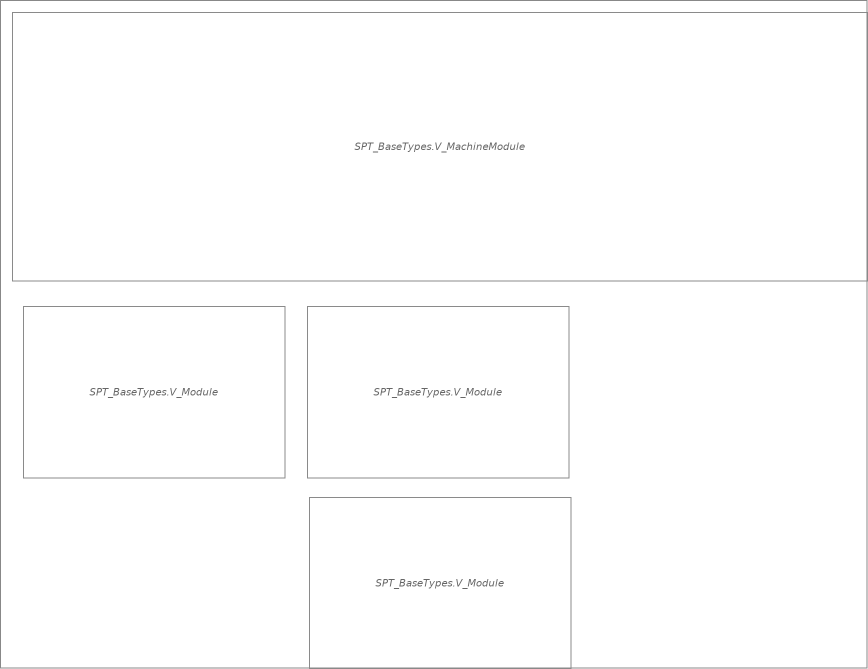
VISUALIZATION Visualization  // 868x669
    Frame (12,12 856x269)
        shows SPT_BaseTypes.V_MachineModule(HMI := MAIN.Machine.PackMLBaseModule_HMI)
    Frame (23,306 262x172)
        shows SPT_BaseTypes.V_Module(HMI := MAIN.Machine.EquipOne.PackMLBaseModule_HMI)
    Frame (307,306 262x172)
        shows SPT_BaseTypes.V_Module(HMI := MAIN.Machine.EquipTwo.PackMLBaseModule_HMI)
    Frame (309,497 262x172)
        shows SPT_BaseTypes.V_Module(HMI := MAIN.Machine.EquipTwo.SubModule.PackMLBaseModule_HMI)
END_VISUALIZATION

(* stored: Version 1.1.0.1, ProductVersion 3.1.4026.12
   Visu Visualization: Id {a30d06ee-a503-46c1-9acf-2579f41ca35a} *)
